INTERFACE I_PersistentEventStorage

METHOD StoreEvent
VAR_INPUT
	stEvent : ST_Event;
END_VAR
END_METHOD

END_INTERFACE

(* stored: Version 1.1.0.1, ProductVersion 3.1.4024.9
   Itf I_PersistentEventStorage: Id {20223271-627b-4152-8c29-c320f20a8be5}
   Method StoreEvent: Id {e7ce9b4c-dfb1-46f4-bf96-d9f7102c1f64} *)
